// TIA Portal V21 export
TYPE "Std_eValveState"
   STRUCT
      NotReady { ExternalVisible := 'False'} : Int := 0;
      Configurable { ExternalVisible := 'False'} : Int := 1;
      Running { ExternalVisible := 'False'} : Int := 2;
      Failure { ExternalVisible := 'False'} : Int := 3;
   END_STRUCT;
END_TYPE
